SUBAPPLICATION Uebung_010d2 (* Toggle Flip-Flop mit IE SoftKey_F1 SK_RELEASED mit GreenWhiteBackground mit Subapp *)
  (* Standard: 61499-2; Description: Copyright (c) 2026 Meisterschulen am Ostbahnhof This program and the accompanying materials are made available under the terms of the Eclipse Public License 2.0 which is available at https://www.eclipse.org/legal/epl-2.0/ SPDX-License-Identifier: EPL-2.0 *)
  (* Version 1.0, 2026-09-02, Franz Höpfinger, Meisterschulen am Ostbahnhof, initial API and implementation and/or initial documentation *)
  PACKAGE Uebungen;
  IMPORT Uebungen::const::UT::DefaultPool::SoftKey_F1;
  IMPORT logiBUS::io::DQ::logiBUS_DO;
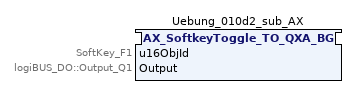
  SUBAPPS
    Uebung_010d2_sub_AX : MyLib::sys::AX_SoftkeyToggle_TO_QXA_BG(u16ObjId := SoftKey_F1 (* Object ID *), Output := logiBUS_DO::Output_Q1 (* Identify the Output Output_Q1..Q8 *));
  END_SUBAPPS
END_SUBAPPLICATION
